{attribute 'qualified_only'}
{attribute 'strict'}
{attribute 'to_string'}
TYPE E_APP_VARIANT :
(
  VARIANT_INVALID,
	VARIANT_OUTPUT_24,
  VARIANT_OUTPUT_CLAMP
);
END_TYPE

(* stored: Version 1.1.0.1
   DUT E_APP_VARIANT: Id {9edcb9a5-412e-4ef9-b1d3-756dd77a4c05} *)
